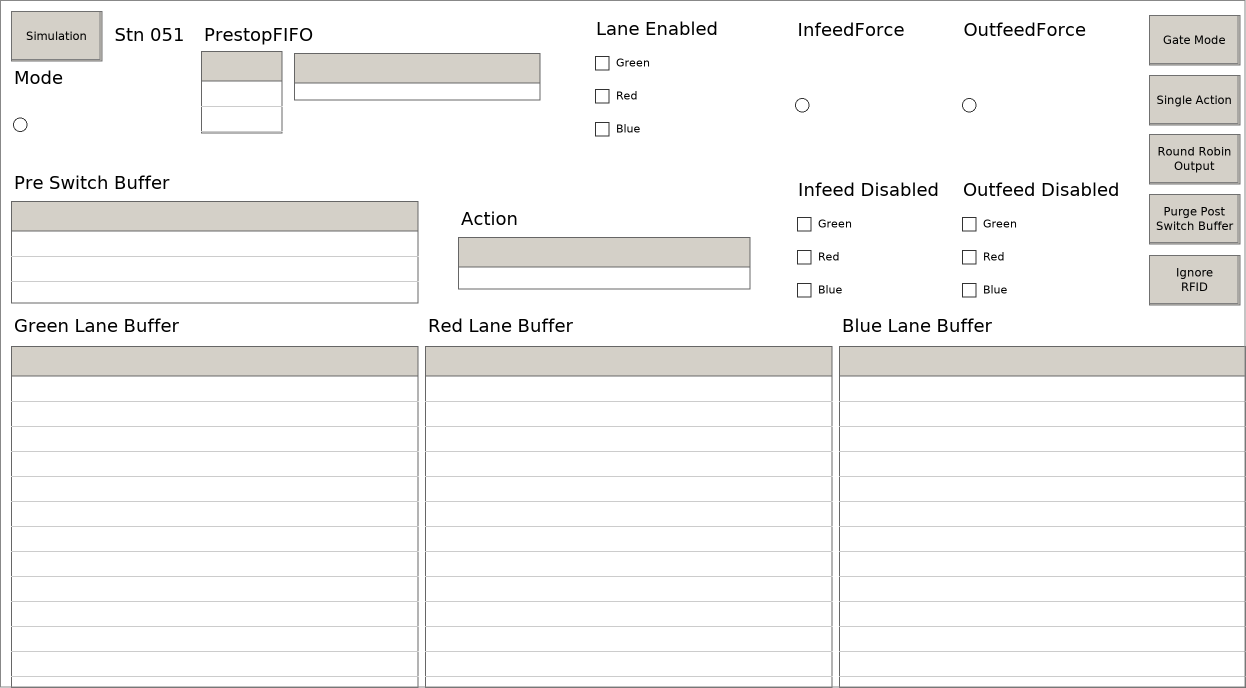
VISUALIZATION ThreeLaneSwitchData  // 1246x688
    Group (11,168 407x135)
        Table (0,33 407x102), data array: Stn051_16_ReturnLnSw.fb3LaneSwitchMain.pCmp^.PreSwitchBuffer
            p3854506369: Stn051_16_ReturnLnSw.fb3LaneSwitchMain.pCmp^.PreSwitchBuffer[INDEX].RFID
            p1892666644: Stn051_16_ReturnLnSw.fb3LaneSwitchMain.pCmp^.PreSwitchBuffer[INDEX].Location
            p338671338: Stn051_16_ReturnLnSw.fb3LaneSwitchMain.pCmp^.PreSwitchBuffer[INDEX].PrimaryLane
            p2170511999: Stn051_16_ReturnLnSw.fb3LaneSwitchMain.pCmp^.PreSwitchBuffer[INDEX].SecondaryLane
            p3723444502: Stn051_16_ReturnLnSw.fb3LaneSwitchMain.pCmp^.PreSwitchBuffer[INDEX].TertiaryLane
            p1218418051: Stn051_16_ReturnLnSw.fb3LaneSwitchMain.pCmp^.PreSwitchBuffer[INDEX].PuckSide
            p746581629: Stn051_16_ReturnLnSw.fb3LaneSwitchMain.pCmp^.PreSwitchBuffer[INDEX].IsHighPriority
            p3104783080: Stn051_16_ReturnLnSw.fb3LaneSwitchMain.pCmp^.PreSwitchBuffer[INDEX].InfeedBelt
            p1755163831: 1st Lane
            p4092479075: 2nd Lane
            p2237128397: 3rd Lane
            p505689113: Puck Side
            p1757482276: High Pr
            p2501879983: Stn051_16_ReturnLnSw.fb3LaneSwitchMain.pCmp^.PreSwitchBuffer[INDEX].OutfeedDivert
            p7306298: Stn051_16_ReturnLnSw.fb3LaneSwitchMain.pCmp^.PreSwitchBuffer[INDEX].TransferStage
        Rectangle (0,0 224x30), "Pre Switch Buffer"
    Table (425,346 407x342), data array: Stn051_16_ReturnLnSw.fb3LaneSwitchMain.pCmp^.PostSwitchBuffer[2]
        p3854506369: Stn051_16_ReturnLnSw.fb3LaneSwitchMain.pCmp^.PostSwitchBuffer[2][INDEX].RFID
        p1892666644: Stn051_16_ReturnLnSw.fb3LaneSwitchMain.pCmp^.PostSwitchBuffer[2][INDEX].Location
        p338671338: Stn051_16_ReturnLnSw.fb3LaneSwitchMain.pCmp^.PostSwitchBuffer[2][INDEX].PrimaryLane
        p2170511999: Stn051_16_ReturnLnSw.fb3LaneSwitchMain.pCmp^.PostSwitchBuffer[2][INDEX].SecondaryLane
        p3723444502: Stn051_16_ReturnLnSw.fb3LaneSwitchMain.pCmp^.PostSwitchBuffer[2][INDEX].TertiaryLane
        p1218418051: Stn051_16_ReturnLnSw.fb3LaneSwitchMain.pCmp^.PostSwitchBuffer[2][INDEX].PuckSide
        p746581629: Stn051_16_ReturnLnSw.fb3LaneSwitchMain.pCmp^.PostSwitchBuffer[2][INDEX].IsHighPriority
        p3104783080: Stn051_16_ReturnLnSw.fb3LaneSwitchMain.pCmp^.PostSwitchBuffer[2][INDEX].InfeedBelt
        p2501879983: Stn051_16_ReturnLnSw.fb3LaneSwitchMain.pCmp^.PostSwitchBuffer[2][INDEX].OutfeedDivert
        p7306298: Stn051_16_ReturnLnSw.fb3LaneSwitchMain.pCmp^.PostSwitchBuffer[2][INDEX].TransferStage
        p1755163831: 1st Lane
        p4092479075: 2nd Lane
        p2237128397: 3rd Lane
        p1757482276: High Pr
    Rectangle (425,311 224x30), "Red Lane Buffer"
    Table (11,346 407x342), data array: Stn051_16_ReturnLnSw.fb3LaneSwitchMain.pCmp^.PostSwitchBuffer[1]
        p3854506369: Stn051_16_ReturnLnSw.fb3LaneSwitchMain.pCmp^.PostSwitchBuffer[1][INDEX].RFID
        p1892666644: Stn051_16_ReturnLnSw.fb3LaneSwitchMain.pCmp^.PostSwitchBuffer[1][INDEX].Location
        p338671338: Stn051_16_ReturnLnSw.fb3LaneSwitchMain.pCmp^.PostSwitchBuffer[1][INDEX].PrimaryLane
        p2170511999: Stn051_16_ReturnLnSw.fb3LaneSwitchMain.pCmp^.PostSwitchBuffer[1][INDEX].SecondaryLane
        p3723444502: Stn051_16_ReturnLnSw.fb3LaneSwitchMain.pCmp^.PostSwitchBuffer[1][INDEX].TertiaryLane
        p1218418051: Stn051_16_ReturnLnSw.fb3LaneSwitchMain.pCmp^.PostSwitchBuffer[1][INDEX].PuckSide
        p746581629: Stn051_16_ReturnLnSw.fb3LaneSwitchMain.pCmp^.PostSwitchBuffer[1][INDEX].IsHighPriority
        p3104783080: Stn051_16_ReturnLnSw.fb3LaneSwitchMain.pCmp^.PostSwitchBuffer[1][INDEX].InfeedBelt
        p2501879983: Stn051_16_ReturnLnSw.fb3LaneSwitchMain.pCmp^.PostSwitchBuffer[1][INDEX].OutfeedDivert
        p7306298: Stn051_16_ReturnLnSw.fb3LaneSwitchMain.pCmp^.PostSwitchBuffer[1][INDEX].TransferStage
        p1755163831: 1st Lane
        p4092479075: 2nd Lane
        p2237128397: 3rd Lane
        p505689113: Puck Side
        p1757482276: High Pr
    Rectangle (11,311 224x30), "Green Lane Buffer"
    Table (839,346 407x342), data array: Stn051_16_ReturnLnSw.fb3LaneSwitchMain.pCmp^.PostSwitchBuffer[3]
        p3854506369: Stn051_16_ReturnLnSw.fb3LaneSwitchMain.pCmp^.PostSwitchBuffer[3][INDEX].RFID
        p1892666644: Stn051_16_ReturnLnSw.fb3LaneSwitchMain.pCmp^.PostSwitchBuffer[3][INDEX].Location
        p338671338: Stn051_16_ReturnLnSw.fb3LaneSwitchMain.pCmp^.PostSwitchBuffer[3][INDEX].PrimaryLane
        p2170511999: Stn051_16_ReturnLnSw.fb3LaneSwitchMain.pCmp^.PostSwitchBuffer[3][INDEX].SecondaryLane
        p3723444502: Stn051_16_ReturnLnSw.fb3LaneSwitchMain.pCmp^.PostSwitchBuffer[3][INDEX].TertiaryLane
        p1218418051: Stn051_16_ReturnLnSw.fb3LaneSwitchMain.pCmp^.PostSwitchBuffer[3][INDEX].PuckSide
        p746581629: Stn051_16_ReturnLnSw.fb3LaneSwitchMain.pCmp^.PostSwitchBuffer[3][INDEX].IsHighPriority
        p3104783080: Stn051_16_ReturnLnSw.fb3LaneSwitchMain.pCmp^.PostSwitchBuffer[3][INDEX].InfeedBelt
        p2501879983: Stn051_16_ReturnLnSw.fb3LaneSwitchMain.pCmp^.PostSwitchBuffer[3][INDEX].OutfeedDivert
        p7306298: Stn051_16_ReturnLnSw.fb3LaneSwitchMain.pCmp^.PostSwitchBuffer[3][INDEX].TransferStage
        p1755163831: 1st Lane
        p4092479075: 2nd Lane
        p2237128397: 3rd Lane
        p505689113: Puck Side
        p1757482276: High Pr
    Rectangle (839,311 224x30), "Blue Lane Buffer"
    Button (1149,15 91x50), "Gate Mode", colour toggle: gStn051_16_ReturnLnSw.Sim.GateActionMode
        toggle gStn051_16_ReturnLnSw.Sim.GateActionMode
    Button (1149,75 91x50), "Single Action", colour toggle: gStn051_16_ReturnLnSw.Sim.GateProceedWithSingleAction
        toggle gStn051_16_ReturnLnSw.Sim.GateProceedWithSingleAction
    Group (793,15 116x151)
        RadioButton (0,29 91x122), variable: gStn051_16_ReturnLnSw.Sim.ForceInfeedLane
            Areas[0]: Text=None
            Areas[1]: Text=Green
            Areas[2]: Text=Red
            Areas[3]: Text=Blue
        Rectangle (0,0 116x30), "InfeedForce"
    Group (960,15 130x151)
        Rectangle (0,0 130x30), "OutfeedForce"
        RadioButton (0,29 91x122), variable: gStn051_16_ReturnLnSw.Sim.ForceOutfeedLane
            Areas[0]: Text=None
            Areas[1]: Text=Green
            Areas[2]: Text=Red
            Areas[3]: Text=Blue
    Button (1149,134 91x50), "Round Robin Output", colour toggle: gStn051_16_ReturnLnSw.Sim.RoundRobinOutput
        toggle gStn051_16_ReturnLnSw.Sim.RoundRobinOutput
    Group (795,175 150x130)
        Rectangle (0,0 147x30), "Infeed Disabled"
        Checkbox (0,34 150x30), "Green", variable: gStn051_16_ReturnLnSw.Sim.InputLaneDisabled[cLaneSel.Green]
        Checkbox (0,67 150x30), "Red", variable: gStn051_16_ReturnLnSw.Sim.InputLaneDisabled[cLaneSel.Red]
        Checkbox (0,100 150x30), "Blue", variable: gStn051_16_ReturnLnSw.Sim.InputLaneDisabled[cLaneSel.Blue]
    Group (960,175 162x130)
        Rectangle (0,0 162x30), "Outfeed Disabled"
        Checkbox (0,34 150x30), "Green", variable: gStn051_16_ReturnLnSw.Sim.OutputLaneDisabled[cLaneSel.Green]
        Checkbox (0,67 150x30), "Red", variable: gStn051_16_ReturnLnSw.Sim.OutputLaneDisabled[cLaneSel.Red]
        Checkbox (0,100 150x30), "Blue", variable: gStn051_16_ReturnLnSw.Sim.OutputLaneDisabled[cLaneSel.Blue]
    Button (1149,194 91x50), "Purge Post Switch Buffer", colour toggle: gStn051_16_ReturnLnSw.Sim.AutoPurgePostSwitch
        toggle gStn051_16_ReturnLnSw.Sim.AutoPurgePostSwitch
    RadioButton (11,91 190x67), variable: gStn051_16_ReturnLnSw.Sim.SimMode
        Areas[0]: Text=No
        Areas[1]: Text=1
        Areas[2]: Text=2
        Areas[3]: Text=3
    Button (11,11 91x50), "Simulation", colour toggle: gSimulateActive
        toggle gSimulateActive
    Rectangle (11,63 58x30), "Mode"
    Button (1149,255 91x50), "Ignore RFID", colour toggle: gStn051_16_ReturnLnSw.Sim.ForceRFID
        toggle gStn051_16_ReturnLnSw.Sim.ForceRFID
    Group (458,204 292x85)
        Table (0,33 292x52), data array: Stn051_16_ReturnLnSw.fb3LaneSwitchMain.Act
            p3854506369: Stn051_16_ReturnLnSw.fb3LaneSwitchMain.Act.OkTo_ReleasePuck
            p1892666644: Stn051_16_ReturnLnSw.fb3LaneSwitchMain.Act.OkTo_Fault
            p338671338: Stn051_16_ReturnLnSw.fb3LaneSwitchMain.Act.Target_Workstop
            p2170511999: Stn051_16_ReturnLnSw.fb3LaneSwitchMain.Act.Target_Lane
            p3723444502: Stn051_16_ReturnLnSw.fb3LaneSwitchMain.Act.Target_FaultCode
            p2232123230: Release Puck
            p1755163831: Work Stop
            p2237128397: Fault #
        Rectangle (0,0 92x30), "Action"
    Group (201,20 339x113)
        Rectangle (0,0 124x30), "PrestopFIFO"
        Table (0,31 81x82), data array: gStn051_16_ReturnLnSw.PrestopFIFO
            p3854506369: gStn051_16_ReturnLnSw.PrestopFIFO[INDEX]
            p2232123230: Lane
        Table (93,33 246x47), data array: Stn051_16_ReturnLnSw.fb3LaneSwitchMain.fbTC.fbTC03.pWorkStop[gStn051_16_ReturnLnSw.PrestopFIFO[0]]^.PuckLnSw
            p3854506369: Stn051_16_ReturnLnSw.fb3LaneSwitchMain.fbTC.fbTC03.pWorkStop[gStn051_16_ReturnLnSw.PrestopFIFO[0]]^.PuckLnSw.RFID
            p1892666644: Stn051_16_ReturnLnSw.fb3LaneSwitchMain.fbTC.fbTC03.pWorkStop[gStn051_16_ReturnLnSw.PrestopFIFO[0]]^.PuckLnSw.Location
            p338671338: Stn051_16_ReturnLnSw.fb3LaneSwitchMain.fbTC.fbTC03.pWorkStop[gStn051_16_ReturnLnSw.PrestopFIFO[0]]^.PuckLnSw.PrimaryLane
            p2170511999: Stn051_16_ReturnLnSw.fb3LaneSwitchMain.fbTC.fbTC03.pWorkStop[gStn051_16_ReturnLnSw.PrestopFIFO[0]]^.PuckLnSw.SecondaryLane
            p3723444502: Stn051_16_ReturnLnSw.fb3LaneSwitchMain.fbTC.fbTC03.pWorkStop[gStn051_16_ReturnLnSw.PrestopFIFO[0]]^.PuckLnSw.TertiaryLane
            p1218418051: Stn051_16_ReturnLnSw.fb3LaneSwitchMain.fbTC.fbTC03.pWorkStop[gStn051_16_ReturnLnSw.PrestopFIFO[0]]^.PuckLnSw.PuckSide
            p746581629: Stn051_16_ReturnLnSw.fb3LaneSwitchMain.fbTC.fbTC03.pWorkStop[gStn051_16_ReturnLnSw.PrestopFIFO[0]]^.PuckLnSw.IsHighPriority
            p3104783080: Stn051_16_ReturnLnSw.fb3LaneSwitchMain.fbTC.fbTC03.pWorkStop[gStn051_16_ReturnLnSw.PrestopFIFO[0]]^.PuckLnSw.InfeedBelt
            p2501879983: Stn051_16_ReturnLnSw.fb3LaneSwitchMain.fbTC.fbTC03.pWorkStop[gStn051_16_ReturnLnSw.PrestopFIFO[0]]^.PuckLnSw.OutfeedDivert
            p7306298: Stn051_16_ReturnLnSw.fb3LaneSwitchMain.fbTC.fbTC03.pWorkStop[gStn051_16_ReturnLnSw.PrestopFIFO[0]]^.PuckLnSw.TransferStage
            p1755163831: 1st Lane
            p4092479075: 2nd Lane
            p2237128397: 3rd Lane
    Rectangle (593,14 162x30), "Lane Enabled"
    Checkbox (593,48 150x30), "Green", variable: gStn051_16_ReturnLnSw.LaneEnabled[cLaneSel.Green]
    Checkbox (593,81 150x30), "Red", variable: gStn051_16_ReturnLnSw.LaneEnabled[cLaneSel.Red]
    Checkbox (593,114 150x30), "Blue", variable: gStn051_16_ReturnLnSw.LaneEnabled[cLaneSel.Blue]
    Label (116,26 67x18), "Stn 051"
END_VISUALIZATION

(* stored: Version 1.1.0.1, ProductVersion 3.1.4024.6
   Visu ThreeLaneSwitchData: Id {23811fc5-5b32-4a4f-94ff-2cd5426aa984} *)
